{attribute 'qualified_only'}
// Robot3 Data-RightArm
VAR_GLOBAL									 
	// absolute encoder value at minimal joint positon
	g_minLinkEncoder :ARRAY[1..g_mArmNum, 1..g_mJntNum] OF DINT :=
		[122745, 128228, 36292, 22430, 2025, 65855, 0,
		 35855, 68924, 4429, 107164, 130111, 62000, 0];
		 
	// absolute encoder value at maximum joint positon
	g_maxLinkEncoder :ARRAY[1..g_mArmNum, 1..g_mJntNum] OF DINT :=
		[36223, 83720, 69818, 109643, 36436, 45700, 0,
		 79841, 24455, 37956, 63571, 31889, 41644, 0];
	
	// absolute encoder value at calibrated positon
	g_caliLinkEncoder :ARRAY[1..g_mArmNum, 1..g_mJntNum] OF DINT :=
		[13129, 106056, 47289, 78598, 85910, 88760, 47232,
		 58523, 46542, 15769, 8255, 81176, 20111, 56205];
	
	 // if absolute encoder value cross zeros within joint motion range
	 // NOTICE: joint 7 is always 0.
	g_linkEncZeroCross :ARRAY[1..g_mArmNum, 1..g_mJntNum] OF INT :=
		[1, 0, 0, 0, 1, 1, 1,
		 0, 0, 1, 1, 0, 1, 1];
		 
	// limit value of gripper hall sensor
	g_minHallSensorValue :ARRAY[1..2] OF DINT:=[9702292,9833247];
	g_maxHallSensorValue :ARRAY[1..2] OF DINT  :=[114690234,115411089];
END_VAR

VAR_GLOBAL CONSTANT	
	
 	//################ DO NOT modify parameters below ###########################	
	// abolute encoder expanded limit buffer in case there is calibrtion error at limit position
	g_linkEncLimitBuffer : DINT := 1000;
	
	// flag if joint can rotate multiple cycles
	g_multipleCyclesJoint :ARRAY[1..g_mArmNum, 1..g_mJntNum] OF INT :=
		[0, 0, 0, 0, 0, 0, 1,
		 0, 0, 0, 0, 0, 0, 1];
		 
	// joint position at link encoder calibrated point
	g_linkEncCaliJntPos :ARRAY[1..g_mArmNum, 1..g_mJntNum] OF LREAL :=
		[0.0, -PI/2, 0.0, -pi, pi, -PI/2, 0.0,
		 0.0, -PI/2, 0.0, 0.0, pi, PI/2, 0.0];

END_VAR

(* stored: Version 1.1.0.1, ProductVersion 3.1.4024.11
   GVL GVL_ArmJointCaliData: Id {110f2ddd-8f6e-45b7-a97a-8030310c3113} *)
